(* IEC 61131-3 sources: lc3-udp/src, 2 files *)

(* ---- types.iecst ---- *)
TYPE
	IPv4Address : ARRAY [0..3] OF BYTE;
	UDPEndpoint : STRUCT
		host : STRING[128];
		port : UINT;
	END_STRUCT;
END_TYPE

(* ---- program.iecst ---- *)
PROGRAM Program1
	VAR
		buffer : ARRAY[0..255] OF BYTE;
		destination : UDPEndpoint;
		bytes_sent : LINT;
	END_VAR

	buffer[0] := 16#BE;
	buffer[1] := 16#EF;
	destination.host := '192.168.1.123';
	destination.port := 1234;

	bytes_sent := sendto(buf := REF(buffer[0]), buflen := SIZEOF(buffer), dst := destination, ENO => ENO);
END_PROGRAM
